// TIA Portal V17 export
// export: Created 2021-12-03T08:12:49.6315421Z, ExportSetting WithDefaults, DisplayName Totally Integrated Automation Portal, DisplayVersion V17, DisplayName TIA Portal Openness, DisplayVersion V17, DisplayName TIA Portal Version Control Interface, DisplayVersion V17, DisplayName STEP 7 Professional, DisplayVersion V17, DisplayName STEP 7 Safety, DisplayVersion V17, DisplayName WinCC Advanced, DisplayVersion V17
FUNCTION "FC_HMI_Communication" : Void   // FC1000, FBD
VERSION : 0.1
// stored: AutoNumber false, IsIECCheckEnabled false, UDAEnableTagReadback false
BEGIN

REGION Network 1
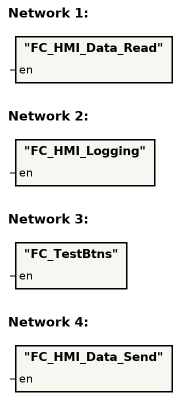
   "FC_HMI_Data_Read"();
END_REGION

REGION Network 2
   "FC_HMI_Logging"();
END_REGION

REGION Network 3
   "FC_TestBtns"();
END_REGION

REGION Network 4
   "FC_HMI_Data_Send"();
END_REGION
END_FUNCTION
